(* PLC project WAVE_TEST, Actility iec61131 1.0.26 *)
(* stored: creationDateTime 2013-01-02T13:55:36, version 1.1.0, modificationDateTime 2013-06-25T12:16:12 *)

PROGRAM Simul_Temperature
  VAR
    Information : STRING := '';
  END_VAR
  VAR_EXTERNAL
    Temperature : REAL;  (* Link to GLOBAL Variable *)
    Global_Config : BOOL;  (* Link to GLOBAL Variable *)
    Global_Resource : BOOL;  (* Link to GLOBAL Variable *)
  END_VAR
  VAR
    AV : REAL := 20;  (* 20 degC *)
    AMP : REAL := 4;  (* from 18 to 22 degC *)
    P : REAL := 30;  (* 30 sec *)
    SIG : INT := 1;  (* Sinus wave *)
    STP : REAL := 20;
    Epsilon : REAL := 0.3;
    V : REAL;
    Wave_Gen : WAVE_GENERATOR;
    Hyst : HYSTERESIS;
  END_VAR

INITIAL_STEP STEP1:
  STEP1_INLINE1(P);
  COMPUTE_FUNCTION_BLOCKS(S);
END_STEP
ACTION STEP1_INLINE1:
  Information:='STEP1 Active';
END_ACTION
TRANSITION FROM STEP1 TO STEP2
  := TRUE;
END_TRANSITION
STEP STEP2:
  STEP2_INLINE2(P);
  Wave_Gen(N);
  Hyst(N);
END_STEP
ACTION STEP2_INLINE2:
  Information:='STEP2 Active';
END_ACTION
TRANSITION FROM STEP2 TO STEP3
  := V = 2.0;
END_TRANSITION
TRANSITION FROM STEP2 TO STEP4
  := V = 1.0;
END_TRANSITION
STEP STEP3:
  STEP3_INLINE3(P);
END_STEP
ACTION STEP3_INLINE3:
  Information:='STEP3 Active';
END_ACTION
TRANSITION FROM STEP3 TO STEP2
  := TRUE;
END_TRANSITION
STEP STEP4:
  STEP4_INLINE4(P);
END_STEP
ACTION STEP4_INLINE4:
  Information:='STEP4 Active';
END_ACTION
TRANSITION FROM STEP4 TO STEP1
  := V=0.0;
END_TRANSITION
ACTION COMPUTE_FUNCTION_BLOCKS:  (* blocks drawn on the SFC sheet *)
  Wave_Gen(Average := AV, Amplitude := AMP, Period := P, SigType := SIG);
  Hyst(XIN1 := Wave_Gen.Value, XIN2 := STP, EPS := Epsilon);
  Temperature := Wave_Gen.Value;
  Global_Config := Hyst.Q;
  Global_Resource := Hyst.Q;
END_ACTION
END_PROGRAM

CONFIGURATION STD_CONF
  VAR_GLOBAL
    Global_Config : BOOL;
    Temperature : REAL := 0.0;  (* Simulated temperature *)
  END_VAR
  RESOURCE STD_RESOURCE ON PLC
    VAR_GLOBAL RETAIN
      Global_Resource : BOOL;
    END_VAR
    TASK STD_TASK(INTERVAL := T#1s0ms, PRIORITY := 0);
    PROGRAM main WITH STD_TASK : Simul_Temperature;
  END_RESOURCE
END_CONFIGURATION
